# EPICS autosave request: streakcameraApp/Db/sc5680.req
$(P)AcqParams:Start-Sel
$(P)CamParams:Exposure-SP
$(P)GenParams:TimeRange-SP
$(P)GenParams:Mode-Sel
$(P)GenParams:GateMode-Sel
$(P)GenParams:MCPGain-SP
$(P)GenParams:Shutter-Sel
$(P)GenParams:BlankingAmp-Sel
$(P)GenParams:HTrigStatus-Sel
$(P)GenParams:HTrigMode-Sel
$(P)GenParams:HTrigLevel-SP
$(P)GenParams:Delay-SP
$(P)GenParams:FocusTimeOver-SP
